(* PLC project PLC, Beckhoff Automation GmbH TwinCAT PLC Control 3.5.13.21 *)
(* stored: creationDateTime 2024-02-17T22:42:53.9472974, modificationDateTime 2024-02-17T22:42:53.9472974 *)

TYPE CylOutput :
STRUCT
	opeFw AT %Q*: BOOL;
	opeRv AT %Q*: BOOL;
END_STRUCT
END_TYPE
